{attribute 'OPC.UA.DA.StructuredType' := '1'}
TYPE ST_eChillerState :
STRUCT
	bError : BOOL;
	bWarning: BOOL;
	//implementation is missing, must be added after startup
END_STRUCT
END_TYPE

(* stored: Version 1.1.0.1, ProductVersion 3.1.4024.9
   DUT ST_eChillerState: Id {f6c1261c-08b2-4bf3-9b97-7dfe1e0ef89d} *)
